Fanuc KAREL source: kx00025.KL

-- PROVISIONAL review KL for V770-1; original PC SHA256 26775c70967cc46657e3233c57d5f1cb0a0010b7c8be540171111ea4d0b87761
-- Incomplete behavior may be omitted. Consult companion uncertainty JSON. Do not deploy.
PROGRAM KX00025
%NOLOCKGROUP
VAR
  I : INTEGER
  J : INTEGER
  B : BOOLEAN
  F : FILE
  S : STRING[80]
-- UNRESOLVED_DECL P type=000102
BEGIN
  -- UNRESOLVED_PC offsets 5-12; opcodes 9D,23
  -- UNRESOLVED_PC offsets 17-21; opcodes 7F
END KX00025
